{attribute 'qualified_only'}
{attribute 'strict'}
{attribute 'to_string'}
TYPE E_BooleanOperator :
(
	ANDop,
	ORop,
	XORop
);
END_TYPE

(* stored: Version 1.1.0.1
   DUT E_BooleanOperator: Id {6b5f3edd-8bef-4788-ae37-170110fd29dc} *)
